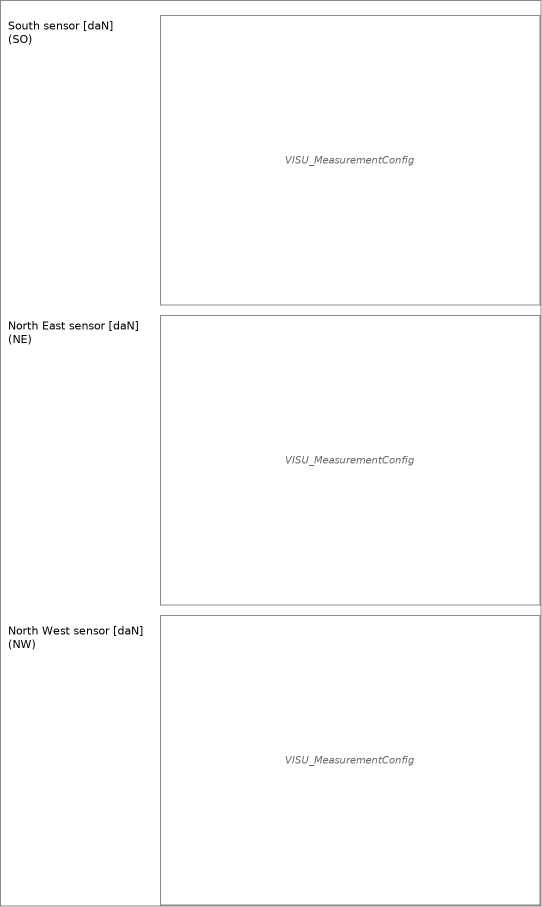
VISUALIZATION VISU_M1Config_Axial_ForceSensors  // 542x907
VAR_IN_OUT
    editable : M1AxialSupportConfig;
	active : M1AxialSupportConfig;
END_VAR
    Label (5,10 180x45), "South sensor [daN] (SO)"
    Label (5,310 145x45), "North East sensor [daN] (NE)"
    Label (5,615 185x45), "North West sensor [daN] (NW)"
    Frame (160,15 380x290)
        shows VISU_MeasurementConfig(active := active.mirrorSouthForce, editable := editable.mirrorSouthForce)
    Frame (160,315 380x290)
        shows VISU_MeasurementConfig(active := active.mirrorNorthEastForce, editable := editable.mirrorNorthEastForce)
    Frame (160,615 380x290)
        shows VISU_MeasurementConfig(active := active.mirrorNorthWestForce, editable := editable.mirrorNorthWestForce)
END_VISUALIZATION

(* stored: Version 1.1.0.1, ProductVersion 3.1.4019.2
   Visu VISU_M1Config_Axial_ForceSensors: Id {747d9d15-7212-41c3-b725-b385997c6f97} *)
